{attribute 'conditionalshow'}
TYPE ST_Var_Info_GV :
STRUCT
	{attribute 'hide'}
	sFullSymbolName				: STRING(48);			//Full Symbol name of plc variable uncoded
	{attribute 'hide'}
	uiSizeArray					: UINT;					//Array size if symbol type is a array
	{attribute 'hide'}
	udiGroup					: UDINT;				//Group number
	{attribute 'hide'}
	udiOffset					: UDINT;				//Offset of group number
	{attribute 'hide'}
	udiSize						: UDINT;				//Size of variable in Byte	
	{attribute 'hide'}
	sSymbolType					: STRING(255);			//Symbol Type
	{attribute 'hide'}
	sSymbolUnit					: STRING(255);			//Comment from the symbol	
END_STRUCT
END_TYPE

(* stored: Version 1.1.0.1, ProductVersion 3.1.4024.6
   DUT ST_Var_Info_GV: Id {32b7120d-3f87-4a6c-963f-c99bd21acce7} *)
